// TIA Portal V20 export
FUNCTION_BLOCK "Tippler_maintenance"   // FB401, LAD
{ S7_Optimized_Access := 'TRUE' }
// stored: AutoNumber false, MemoryReserve 100, SetENOAutomatically false
   VAR_INPUT
      hmi_arm_selection : Int;
      hmi_button_up : Bool;
      hmi_button_down : Bool;
      hmi_set_angle : Int;
      Arm_1_Angle_Value : Real;
      Arm_2_Angle_Value : Real;
      hmi_button_open : Bool;
      hmi_button_close : Bool;
   END_VAR
   VAR_OUTPUT
      Arm1 : Int;
      Arm2 : Int;
      closeUpperClamp : Bool;
      openUpperClamp : Bool;
      closeLowerClamp : Bool;
      openLowerClamp : Bool;
   END_VAR
   VAR
      Arm1SetPosReached : Bool;
      Arm2SetPosReached : Bool;
      speed : Int;
   END_VAR
BEGIN

REGION Network 1 (SCL): Manual operating
   #Arm1 := 0;
   #Arm2 := 0;
   #speed := 0;
   IF #Arm_1_Angle_Value > 50 OR #Arm_2_Angle_Value > 50 THEN
       #speed := 15000;
   ELSE
       #speed := 20000;
   END_IF;
   IF #hmi_arm_selection = 1 THEN
       IF #hmi_button_up AND #hmi_set_angle > #Arm_1_Angle_Value THEN
           #Arm1 :=#speed;
           #Arm2 := 0;
           #closeUpperClamp := FALSE;
           #closeLowerClamp := FALSE;
           #openUpperClamp := FALSE;
           #openLowerClamp := FALSE;
       ELSIF #hmi_button_down THEN
           #Arm1 := -#speed;
           #Arm2 := 0;
           #closeUpperClamp := FALSE;
           #closeLowerClamp := FALSE;
           #openUpperClamp := FALSE;
           #openLowerClamp := FALSE;
       ELSIF #hmi_button_close THEN
           #Arm1 := 0;
           #Arm2 := 0;
           #closeUpperClamp := TRUE;
           #closeLowerClamp := FALSE;
           #openUpperClamp := FALSE; 
           #openLowerClamp := FALSE;
       ELSIF #hmi_button_open THEN
           #Arm1 := 0;
           #Arm2 := 0;
           #closeUpperClamp := FALSE;
           #closeLowerClamp := FALSE;
           #openUpperClamp := TRUE;
           #openLowerClamp := FALSE;
       ELSE
           #Arm1 := 0;
           #Arm2 := 0;
           #closeUpperClamp := FALSE;
           #closeLowerClamp := FALSE;
           #openUpperClamp := FALSE;
           #openLowerClamp := FALSE;
       END_IF;
   ELSIF #hmi_arm_selection = 2  THEN
       IF #hmi_button_up AND #hmi_set_angle > #Arm_2_Angle_Value THEN
           #Arm2 := #speed;
           #Arm1 := 0;
           #closeUpperClamp := FALSE;
           #closeLowerClamp := FALSE;
           #openUpperClamp := FALSE;
           #openLowerClamp := FALSE;
       ELSIF #hmi_button_down THEN
           #Arm2 := -#speed;
           #Arm1 := 0;
           #closeUpperClamp := FALSE;
           #closeLowerClamp := FALSE;
           #openUpperClamp := FALSE;
           #openLowerClamp := FALSE;
       ELSIF #hmi_button_close THEN
           #Arm1 := 0;
           #Arm2 := 0;
           #closeUpperClamp := FALSE;
           #closeLowerClamp := TRUE;
           #openUpperClamp := FALSE;
           #openLowerClamp := FALSE;
       ELSIF #hmi_button_open THEN
           #Arm1 := 0;
           #Arm2 := 0;
           #closeUpperClamp := FALSE;
           #closeLowerClamp := FALSE;
           #openUpperClamp := FALSE;
           #openLowerClamp := TRUE;
       ELSE
           #Arm2 := 0;
           #Arm1 := 0;
           #closeUpperClamp := FALSE;
           #closeLowerClamp := FALSE;
           #openUpperClamp := FALSE;
           #openLowerClamp := FALSE;
       END_IF;
   ELSIF #hmi_arm_selection = 0 THEN
       IF #hmi_button_up THEN
           IF #hmi_set_angle > #Arm_2_Angle_Value AND #hmi_set_angle > #Arm_1_Angle_Value THEN
               #Arm1 := #speed;
               #Arm2 := #speed;
               #closeUpperClamp := FALSE;
               #closeLowerClamp := FALSE;
               #openUpperClamp := FALSE;
               #openLowerClamp := FALSE;
           ELSIF #hmi_set_angle > #Arm_2_Angle_Value AND #hmi_set_angle < #Arm_1_Angle_Value THEN
               #Arm1 := 0;
               #Arm2 := #speed;
               #closeUpperClamp := FALSE;
               #closeLowerClamp := FALSE;
               #openUpperClamp := FALSE;
               #openLowerClamp := FALSE;
           ELSIF #hmi_set_angle < #Arm_2_Angle_Value AND #hmi_set_angle > #Arm_1_Angle_Value THEN
               #Arm1 := #speed;
               #Arm2 := 0;
               #closeUpperClamp := FALSE;
               #closeLowerClamp := FALSE;
               #openUpperClamp := FALSE;
               #openLowerClamp := FALSE;
           ELSE
               #Arm1 := 0;
               #Arm2 := 0;
               #closeUpperClamp := FALSE;
               #closeLowerClamp := FALSE;
               #openUpperClamp := FALSE;
               #openLowerClamp := FALSE;
           END_IF;
       ELSIF #hmi_button_down THEN
           #Arm2 := -#speed;
           #Arm1 := -#speed;
           #closeUpperClamp := FALSE;
           #closeLowerClamp := FALSE;
           #openUpperClamp := FALSE;
           #openLowerClamp := FALSE;
       ELSIF #hmi_button_close THEN
           #Arm1 := 0;
           #Arm2 := 0;
           #closeUpperClamp := TRUE;
           #closeLowerClamp := TRUE;
           #openUpperClamp := FALSE;
           #openLowerClamp := FALSE;
       ELSIF #hmi_button_open THEN
           #Arm1 := 0;
           #Arm2 := 0;
           #closeUpperClamp := FALSE;
           #closeLowerClamp := FALSE;
           #openUpperClamp := TRUE;
           #openLowerClamp := TRUE;
       ELSE
           #Arm2 := 0;
           #Arm1 := 0;
           #closeUpperClamp := FALSE;
           #closeLowerClamp := FALSE;
           #openUpperClamp := FALSE;
           #openLowerClamp := FALSE;
       END_IF;
   ELSE
       #Arm1 := 0;
       #Arm2 := 0;
       #closeUpperClamp := FALSE;
       #closeLowerClamp := FALSE;
       #openUpperClamp := FALSE;
       #openLowerClamp := FALSE;
   END_IF;
END_REGION

REGION Network 2 (SCL)
   IF #Arm_1_Angle_Value > #hmi_set_angle THEN
       #Arm1SetPosReached := 1;

   ELSE
       #Arm1SetPosReached := 0;
   END_IF;
   IF #Arm_2_Angle_Value > #hmi_set_angle THEN
       #Arm2SetPosReached := 1;
   ELSE
       #Arm2SetPosReached := 0;
   END_IF;
END_REGION
END_FUNCTION_BLOCK
